INTERFACE I_Timer

METHOD Execute
END_METHOD

METHOD Register
END_METHOD

END_INTERFACE

(* stored: Version 1.1.0.1, ProductVersion 3.1.4024.10
   Itf I_Timer: Id {9ac5e8ce-e818-4c15-a668-07abdcf7a410}
   Method Execute: Id {06a442e1-fad7-4217-84f9-25bf203c3a8a}
   Method Register: Id {eb5135c7-2316-425f-8c27-94d145cf86e7} *)
